# B&R Automation Studio project BuR
Automation Studio 4.5.2.102

## Logical view

### Package Logical/Libraries - Global libraries

### Library Logical/Libraries/DebuggingCom/DebComLib (IEC, version 1.00.1)
Depends on: astime, AsBrStr, TCPComLib

#### Types.typ - Exported data types
```iecst
TYPE
	e_DebugDataType : (E_STRING
		,E_DATA
	);

	e_DebugStepSend : (STEP_WAIT_FOR_ACTIVATE,
		STEP_WAIT_FOR_SEND_REQ,
		STEP_WAIT_FOR_ACK
	);

	s_SendDataType : STRUCT
		Data : ARRAY [0..ui_Max_Send_DataSize] OF BYTE;
		ui_Size : UINT;
	END_STRUCT;

	s_DebugDataType : STRUCT
		e_DataType : e_DebugDataType;
		ui_DataSize : UINT;
		(* *)
		tod_Time : TOD;
		dt_Date : DATE;
		str_Description : STRING[80];
		i_DataType : INT;
		aby_Data : ARRAY[0..ui_Data_Length_Pure_Data] OF BYTE;
    END_STRUCT;

	s_DebugDataBufferType : STRUCT
		Data : ARRAY[0..ui_Buffer_Size] OF s_DebugDataType;
        Size : INT := 0;
        Index : INT := 0;
	END_STRUCT;

    s_DebuggingComType : STRUCT
        b_init : BOOL := TRUE; (* Initialisierung *)
        b_Connected : BOOL;
        b_Error : BOOL;
        b_Enable_Com : BOOL := TRUE;
        Data : s_DebugDataBufferType;
        AddString : Add_Debug_String;
        AddData : Add_Debug_Data;
        TempStr : STRING[80];
        TempStr2 : STRING[80];
        Internal : s_DebugIternalType;
    END_STRUCT;

  s_DebugIternalType : STRUCT
    Cyclic : CyclicOperations;
  END_STRUCT;
END_TYPE
```

#### Constants.var - Exported constants
```iecst
VAR CONSTANT
	ui_Header_Length            : UINT := 6;          (* STX(1) + Laufnummer(1) + Trennbyte(1) + Telegrammtyp(2) + Trennbyte(1) *)
	ui_Footer_Length            : UINT := 1;          (* ETX(1) *)
	ui_Data_Length_String       : UINT := 90;         (* Zeit(4) + Trennbyte(1) + Datum(4) + Trennbyte(1) + Text(80) *)
	ui_Data_Length_Data         : UINT := 1449;       (* Zeit(4) + Trennbyte(1) + Datum(4) + Trennbyte(1) + Text(80) + Trennbyte(1) + Datentyp(2) + Trennbyte(1) + Daten(1355) *)
	ui_Data_Length_Pure_Data    : UINT := 1355;

	ui_SendDataLength_Debug     : UINT := ui_Header_Length + ui_Data_Length_String + ui_Footer_Length;
	ui_SendDataLength_Data      : UINT := ui_Header_Length + ui_Data_Length_Data + ui_Footer_Length;
	ui_RecDataLength_Quit       : UINT := ui_Header_Length + ui_Footer_Length; (* Quittierung erfolgt über Telegrammnummer *)

	ui_Max_Send_DataSize        : UINT := ui_SendDataLength_Data; (* Muss gröster Datenlänge entsprechen die gesendet werden soll *)

	ui_Buffer_Size              : UINT := 200; (* Größe des in der Steuerung gehaltenen Logs *)
END_VAR
```

#### DebComLib.fun - Exported functions and function blocks
```iecst
FUNCTION_BLOCK CyclicOperations (* *) (*$GROUP=User,$CAT=User,$GROUPICON=User.png,$CATICON=User.png*)
	VAR_INPUT
		Instance : REFERENCE TO s_DebuggingComType;
	END_VAR
	VAR
		FB_DebugCom : FBCom;
		DebugComConfig : s_FBComConfigType;
		FB_ConvertHeader    : ConvertHeader         ;
		FB_ConvertReceivedata : ConvertReceiveData  ;
		b_Enable           : BOOL                   ;
		b_Communicate       : BOOL  := FALSE        ;
		b_DataReceived       : BOOL                 ;
		b_AbortCommunication: BOOL                  ;
		b_Acknowledge      : BOOL                   ;
		b_Enable_Timeout   : BOOL                   ;
		b_Sending           : BOOL                  ;
		b_Wait_Ack          : BOOL                  ;
		b_Packet_Quit       : BOOL                  ;
		b_Data_Fail         : BOOL                  ;
		u16SendDataLength   : UINT                  ;
		u16ReceivedLength   : UDINT                 ;
		ui_pointer          : DINT                  ;
		ui_Packet_Length    : UINT                  ;
		ui_pointer_Data_in  : UINT                  ;
		i_Send_Versuche     : INT                   ;
		i_Rec_Versuche      : INT                   ;
		usi_Lfd_Nr_Send      : USINT                  ;
		usi_Lfd_Nr_Rec       : USINT                  ;
		rt_Count_Send       : R_TRIG                ;
        ton_SendCycle       : TON                   ;
        i_Temp              : INT                   ;

		e_StepSend         : e_DebugStepSend        ;
		e_OldStepSend      : e_DebugStepSend        ;

		aby_SendBuffer : ARRAY [0..ui_Max_Send_DataSize] OF BYTE;
		aby_ReceiveBuffer : ARRAY [0..ui_RecDataLength_Quit] OF BYTE;
		aby_TempBuffer : ARRAY [0..ui_RecDataLength_Quit] OF BYTE;
		aby_Temp : ARRAY[0..ui_Max_Send_DataSize] OF BYTE;
	END_VAR
END_FUNCTION_BLOCK

FUNCTION_BLOCK Add_Debug_String (*//======= Add_Debug_String ===========================================================
// Funktion         : Diese Funktion fügt einen neuen Text und die aktuelle Zeit zum Puffer hinzu
//
// Eingansparameter :
//               str_Text            : zu schreibender Text (STRING[80])
//
// Rückgabewert :
//
// Unterprogramme   : keine
//
// Benötigte Units  :
//
// Aenderungen      :
//
// Aenderungsdatum  :
//
//----------------------------------------------------------------------------------------*) (*$GROUP=User,$CAT=User,$GROUPICON=User.png,$CATICON=User.png*)
	VAR_INPUT
		Instance : REFERENCE TO s_DebuggingComType;
		str_Text : STRING[80];
	END_VAR
	VAR
        realtime : DTStructureGetTime;
		ActTime : DTStructure;
	END_VAR
END_FUNCTION_BLOCK

FUNCTION_BLOCK Add_Debug_Data (*//======= Add_Debug_Data ===========================================================
// Funktion         : Diese Funktion fügt einen neuen Text, neue Daten und die aktuelle Zeit zum Puffer hinzu
//
// Eingansparameter :
//               str_Text            : zu schreibender Text (STRING[80])
//               i_DataType          : Datentyp in aby_Data (INT)
//               aby_Data            : Daten (ARRAY[0..1372] OF BYTE)
//               ui_DataSize         : Länge der übergebenen Daten (UINT)
//
// Rückgabewert :
//
// Unterprogramme   : keine
//
// Benötigte Units  :
//
// Aenderungen      :
//
// Aenderungsdatum  :
//
//----------------------------------------------------------------------------------------*) (*$GROUP=User,$CAT=User,$GROUPICON=User.png,$CATICON=User.png*)
	VAR_INPUT
		Instance : REFERENCE TO s_DebuggingComType;
		str_Text : STRING[80];
		i_DataType : INT;
		aby_Data : ARRAY[0..ui_Data_Length_Pure_Data] OF BYTE;
		ui_DataSize : UINT;
	END_VAR
	VAR
        realtime : DTStructureGetTime;
		ActTime : DTStructure;
	END_VAR
END_FUNCTION_BLOCK

FUNCTION MakeData : USINT
	(*//======= MakeData ===========================================================
	// Funktion         : Diese Funktion konvertiert den Debugtext in ein Bytearray
	//
	// Eingansparameter :
	//
	// Durchgangsparameter :
	//               Data            : Datengrundlage (s_DebugDataType)
	//           aby_Result          : Ergebnis (ARRAY[0..ui_Max_Send_DataSize-1] OF BYTE)
	//
	// Rückgabewert :
	//
	// Unterprogramme   : keine
	//
	// Benötigte Units  :
	//
	// Aenderungen      :
	//
	// Aenderungsdatum  :
	//
	//----------------------------------------------------------------------------------------*)

	VAR_IN_OUT
		Data : s_DebugDataType; (* Datengrundlage *)
		aby_Result : ARRAY[0..ui_Max_Send_DataSize] OF BYTE; (* Ergebnis *)
	END_VAR

	VAR
		i_Temp : INT;
		by_Temp : BYTE;
		tod_Temp : TIME_OF_DAY;
		udi_Temp : UDINT;
	END_VAR

		END_FUNCTION

FUNCTION GetNextTelegramNo : USINT
	VAR_IN_OUT
		usi_ActNo : USINT;
	END_VAR
		END_FUNCTION

FUNCTION MakeSendData : USINT
	(*//======= MakeSendData ===========================================================
	// Funktion         : Diese Funktion setzt den Header und Footer an die Nutdaten
	//
	// Eingansparameter :
	//               ui_DataLength      : genutzte Übergabedatenlänge (UINT)
	//               usi_lfd_Nr         : Telegrammlaufnummer (USINT)
	//
	// Durchgangsparameter :
	//               aby_SourceData     : Datenarray (ARRAY[0..ui_Max_Send_DataSize] OF BYTE)
	//               aby_Result         : Datenarray (ARRAY[0..ui_Max_Send_DataSize - 1] OF BYTE)
	//
	// Rückgabewert :
	//
	// Unterprogramme   : keine
	//
	// Benötigte Units  :
	//
	// Aenderungen      :
	//
	// Aenderungsdatum  :
	//
	//----------------------------------------------------------------------------------------*)
	VAR_INPUT
		ui_DataLength : UINT;
		usi_lfd_Nr : USINT;
		i_TelegrammType : INT;
	END_VAR

	VAR_IN_OUT
		aby_SourceData : ARRAY[0..ui_Max_Send_DataSize] OF BYTE;
		aby_Result : ARRAY[0..ui_Max_Send_DataSize] OF BYTE;
	END_VAR

	VAR
		by_Temp     : BYTE;
		i_Temp : INT;
	END_VAR
			END_FUNCTION

FUNCTION_BLOCK ConvertHeader
	(*//======= ConvertHeader ===========================================================
	// Funktion         : Dieser Funktionsbaustein prüft die empfangenen Headerdaten
	//                 Gibt notwendige Headerdaten aus
	//
	// Eingansparameter :
	//
	// Ein- Ausgansparameter :
	//                   aby_SourceData     : Datenarray (ARRAY[0..ui_RecDataLength_Quit] OF BYTE)
	//
	// Ausgangsparameter:
	//             usi_lfd_Nr_Rec       : Telegrammlaufnummer (USINT)
	//             i_Telegramm_Nr       : Nummer des empfangenen Telegramms (INT)
	//             ui_TotalDataLength   : erwartete Gesammtdatenmenge (UINT)
	//             b_Data_Ok            : Daten Ok (BOOL)
	//
	// Unterprogramme   : keine
	//
	// Benötigte Units  :
	//
	// Aenderungen      :
	//
	// Aenderungsdatum  :
	//
	//----------------------------------------------------------------------------------------*)
	VAR_IN_OUT
		aby_SourceData : ARRAY[0..ui_RecDataLength_Quit] OF BYTE;
	END_VAR

	VAR_OUTPUT
		usi_lfd_Nr_Rec : USINT;
		i_Telegramm_Nr : INT;
		ui_TotalDataLength : UINT;
		b_Data_Ok : BOOL;
	END_VAR

	VAR
		i_Temp : INT;
	END_VAR

		END_FUNCTION_BLOCK

FUNCTION_BLOCK ConvertReceiveData
	(*//======= ConvertReceiveData ===========================================================
	// Funktion         : Dieser Funktionsbaustein prüft die empfangenen Daten
	//                 Entfernt Header und Footer
	//                 Gibt notwendige Daten aus
	//
	//
	// Eingansparameter :
	//               ui_DataLength      : übergebene Nutzdatenlänge (UINT)
	//               i_Telegramm_Nr       : Nummer des empfangenen Telegramms (INT)
	//
	// Ein- Ausgansparameter :
	//
	// Ausgangsparameter:
	//               b_Data_Ok          : Daten sind ok (BOOL);
	//
	//
	// Unterprogramme   : keine
	//
	// Benötigte Units  :
	//
	// Aenderungen      :
	//
	// Aenderungsdatum  :
	//
	//----------------------------------------------------------------------------------------*)
	VAR_INPUT
		ui_DataLength : UINT;
		i_Telegramm_Nr : INT;
	END_VAR

	VAR_OUTPUT
		b_Data_Ok : BOOL;
	END_VAR

		END_FUNCTION_BLOCK
```

#### CyclicOperations.st
```iecst
(* TODO: Hier einen Kommentar eingeben *)
FUNCTION_BLOCK CyclicOperations

	IF Instance.b_init THEN
		DebugComConfig.Connection.b_IsClient := FALSE;
		DebugComConfig.Connection.ui_LocalPort := 5000;
		usi_Lfd_Nr_Send := 0;
		i_Send_Versuche := 0;
		i_Rec_Versuche := 0;

		Instance.b_init := FALSE;
	END_IF;

	CASE e_StepSend OF

		STEP_WAIT_FOR_ACTIVATE:

			IF b_AbortCommunication THEN
				b_AbortCommunication  := FALSE;
			END_IF;

			b_Acknowledge := FALSE;
			b_Communicate := FALSE;
			usi_Lfd_Nr_Send := 0;

			IF b_Enable AND Instance.b_Connected THEN
				e_StepSend := STEP_WAIT_FOR_SEND_REQ;
			END_IF;

		STEP_WAIT_FOR_SEND_REQ:

			// Flankenerzeugung
			b_Communicate      := FALSE;
			b_Acknowledge      := FALSE;

			IF NOT b_Enable THEN
				// Kommunikation deaktivieren

				e_StepSend := STEP_WAIT_FOR_ACTIVATE;
			ELSIF NOT Instance.b_Connected THEN
				// Verbindung wurde geschlossen

				e_StepSend := STEP_WAIT_FOR_ACTIVATE;
			ELSIF b_AbortCommunication THEN
				b_AbortCommunication  := FALSE;
				b_Acknowledge := FALSE;

			ELSE
                IF NOT b_Sending AND NOT b_Communicate AND NOT b_Wait_Ack AND Instance.Data.Size > 0 THEN
                    i_Temp := (Instance.Data.Index + (-(Instance.Data.Size) + ui_Buffer_Size)) MOD ui_Buffer_Size;
                    MakeData(
					Data := Instance.Data.Data[i_Temp]
					,aby_Result := aby_Temp
					);

					IF Instance.Data.Data[i_Temp].e_DataType = E_STRING THEN
						MakeSendData(
							ui_DataLength := ui_Data_Length_String
							,usi_lfd_Nr := GetNextTelegramNo(usi_Lfd_Nr_Send)
							,i_TelegrammType := 16#3032
							,aby_SourceData := aby_Temp
							,aby_Result := aby_SendBuffer
							);
						u16SendDataLength := ui_SendDataLength_Debug;
					ELSE
						MakeSendData(
							ui_DataLength := ui_Data_Length_Data
							,usi_lfd_Nr := GetNextTelegramNo(usi_Lfd_Nr_Send)
							,i_TelegrammType := 16#3033
							,aby_SourceData := aby_Temp
							,aby_Result := aby_SendBuffer
							);
						u16SendDataLength := ui_SendDataLength_Data;
					END_IF;

					b_Communicate := TRUE;
					b_Wait_Ack := TRUE;

					Instance.Data.Size := Instance.Data.Size - 1;

					e_StepSend := STEP_WAIT_FOR_ACK;
				ELSIF b_Wait_Ack THEN
					b_Communicate := TRUE;

					e_StepSend := STEP_WAIT_FOR_ACK;
				END_IF;
			END_IF;

		STEP_WAIT_FOR_ACK:

			// Flankenerzeugung
			b_Communicate := FALSE;

			IF ton_SendCycle.Q THEN
				b_Communicate := TRUE;
			END_IF;

			IF NOT b_Enable THEN
				// Kommunikation deaktivieren

				e_StepSend := STEP_WAIT_FOR_ACTIVATE;
			ELSIF b_AbortCommunication THEN
				// aktuellen Übertragungsvorgang abbrechen

				e_StepSend := STEP_WAIT_FOR_SEND_REQ;
			ELSIF NOT Instance.b_Connected THEN
				// Verbindung wurde geschlossen

				e_StepSend := STEP_WAIT_FOR_ACTIVATE;
			ELSE
				// Quittung empfangen -> auswerten
				IF b_Packet_Quit THEN
					b_Acknowledge := TRUE;
					b_Wait_Ack := FALSE;
					b_Packet_Quit := FALSE;

					e_StepSend := STEP_WAIT_FOR_SEND_REQ;
				END_IF;

			END_IF;

		ELSE
			;
	END_CASE;

	// Timer für zyklisches "Neu-Senden", falls keine Quittung innerhalb der konfigurierten Wartezeit kommt
	b_Enable_Timeout := (e_StepSend = STEP_WAIT_FOR_ACK) AND
	e_StepSend = e_OldStepSend;

	ton_SendCycle (IN := b_Enable_Timeout AND NOT b_Communicate AND NOT ton_SendCycle.Q, PT := t#2000ms);
	e_OldStepSend := e_StepSend;

	// Zähler Sendeversuche
	rt_Count_Send (CLK := b_Sending AND e_StepSend = STEP_WAIT_FOR_ACK); // Flanke zählen Sendeversuche

	// Zähler Rücksetzen
	IF b_Acknowledge OR NOT b_Enable THEN
		i_Send_Versuche := 0;
	END_IF;

	// Zähler Empfangsversuche
	IF b_Data_Fail THEN
		i_Rec_Versuche := i_Rec_Versuche + 1;
	END_IF;

	// Zähler Rücksetzen
	IF NOT b_Enable THEN
		i_Rec_Versuche := 0;
	END_IF;

	IF Instance.b_Enable_Com AND NOT Instance.b_init AND i_Send_Versuche <= 3 AND i_Rec_Versuche <= 3 AND NOT FB_DebugCom.error THEN
		b_Enable := TRUE ;
	ELSE
		b_Enable := FALSE ;
		ui_pointer_Data_in := 0;
	END_IF ;

	//call communication function block
	FB_DebugCom(
		enable := b_Enable
		,send := b_Communicate
		,sendDataLength := u16SendDataLength
		,receiveDataLength := SIZEOF(aby_ReceiveBuffer)
		,configurations := DebugComConfig
		,sendBuffer := ADR(aby_SendBuffer)
		,receiveBuffer := ADR(aby_ReceiveBuffer)
	);
	u16ReceivedLength := FB_DebugCom.receivedDataLength;
	Instance.b_Connected := FB_DebugCom.connected;
	b_DataReceived := FB_DebugCom.dataReceived;
	b_Sending := FB_DebugCom.sending;

	b_Data_Fail := FALSE;

	IF Instance.b_Connected THEN
		// Wenn richtige Datenlänge empfangen und in Speicher eintragen
		IF b_DataReceived THEN
			FOR ui_pointer := 0 TO UDINT_TO_DINT(u16ReceivedLength) - 1 DO

				aby_TempBuffer[ui_pointer_Data_in] := aby_ReceiveBuffer[ui_pointer] ;
				ui_pointer_Data_in := ui_pointer_Data_in + 1;

				IF ui_pointer_Data_in = ui_Header_Length THEN
					FB_ConvertHeader(
						aby_SourceData := aby_TempBuffer
						//,usi_Lfd_Nr_Rec =>
						// ,i_Telegramm_Nr =>
						//,ui_TotalDataLength =>
						// ,b_Data_Ok
						);
					usi_Lfd_Nr_Rec := FB_ConvertHeader.usi_lfd_Nr_Rec;
					ui_Packet_Length := FB_ConvertHeader.ui_TotalDataLength;
				END_IF;

				// Unbekannte Telegrammnummer
				IF ui_pointer_Data_in = ui_Header_Length AND NOT FB_ConvertHeader.b_Data_Ok THEN
					b_Data_Fail := TRUE;
					ui_pointer_Data_in := 0;
				END_IF;

				IF ui_pointer_Data_in = ui_Packet_Length AND ui_pointer_Data_in > ui_Header_Length THEN
					IF aby_TempBuffer[ui_pointer_Data_in - 1] = 16#03 THEN
						// Ende Datenstream
						FB_ConvertReceivedata(
							ui_DataLength := ui_Packet_Length
						,i_Telegramm_Nr := FB_ConvertHeader.i_Telegramm_Nr
						// ,b_Data_Ok =>
						);
						CASE FB_ConvertReceivedata.i_Telegramm_Nr OF

							11: b_Packet_Quit := FB_ConvertHeader.b_Data_Ok AND FB_ConvertReceivedata.b_Data_Ok;

							12: b_Packet_Quit := FB_ConvertHeader.b_Data_Ok AND FB_ConvertReceivedata.b_Data_Ok;

							13: b_Packet_Quit := FB_ConvertHeader.b_Data_Ok AND FB_ConvertReceivedata.b_Data_Ok;

						END_CASE;
						ui_pointer_Data_in := 0 ;
						i_Rec_Versuche := 0;
					ELSE
						ui_pointer_Data_in := 0 ;
						b_Data_Fail := TRUE;
					END_IF;
				END_IF;
			END_FOR ;
		END_IF ;
	ELSE
		ui_pointer_Data_in := 0 ;
	END_IF;

END_FUNCTION_BLOCK
```

#### AddDebugString.st
```iecst
FUNCTION_BLOCK Add_Debug_String
    realtime(enable := TRUE, pDTStructure := ADR(ActTime));
    Instance.Data.Data[Instance.Data.Index].e_DataType := E_STRING;
    Instance.Data.Data[Instance.Data.Index].ui_DataSize := 0;
    Instance.Data.Data[Instance.Data.Index].tod_Time := DT_TO_TOD(DTStructure_TO_DT(ADR(ActTime))) + UINT_TO_TIME(ActTime.millisec);
    Instance.Data.Data[Instance.Data.Index].dt_Date := DT_TO_DATE(DTStructure_TO_DT(ADR(ActTime)));
    Instance.Data.Data[Instance.Data.Index].str_Description := str_Text;
    Instance.Data.Data[Instance.Data.Index].i_DataType := -1;
    Instance.Data.Index := (Instance.Data.Index + 1) MOD ui_Buffer_Size;
    Instance.Data.Size :=  MIN(Instance.Data.Size + 1, UINT_TO_INT(ui_Buffer_Size));
END_FUNCTION_BLOCK
```

#### AddDebugData.st
```iecst
FUNCTION_BLOCK Add_Debug_Data
	realtime(enable := TRUE, pDTStructure := ADR(ActTime));
    Instance.Data.Data[Instance.Data.Index].e_DataType := E_DATA;
	Instance.Data.Data[Instance.Data.Index].ui_DataSize := MIN(ui_DataSize, ui_Data_Length_Pure_Data) ;
	Instance.Data.Data[Instance.Data.Index].tod_Time := DT_TO_TOD(DTStructure_TO_DT(ADR(ActTime))) + UINT_TO_TIME(ActTime.millisec);
	Instance.Data.Data[Instance.Data.Index].dt_Date := DT_TO_DATE(DTStructure_TO_DT(ADR(ActTime)));
	Instance.Data.Data[Instance.Data.Index].str_Description := str_Text;
	Instance.Data.Data[Instance.Data.Index].i_DataType := i_DataType;
	Instance.Data.Data[Instance.Data.Index].aby_Data := aby_Data;
    Instance.Data.Index := (Instance.Data.Index + 1) MOD ui_Buffer_Size;
    Instance.Data.Size :=  MIN(Instance.Data.Size + 1, UINT_TO_INT(ui_Buffer_Size));
END_FUNCTION_BLOCK
```

#### InternalFunctions.st
```iecst
FUNCTION MakeData
	// Reset memory data
	brsmemset(ADR(aby_Result[0]), 0, SIZEOF(aby_Result));
	// Zeit
	tod_Temp := swapTOD(H_TO_NTOD(Data.tod_Time));
	brsmemcpy(ADR(aby_Result[0]), ADR(tod_Temp), SIZEOF(tod_Temp));
	// Trennbyte
	by_Temp := 16#2e;
	brsmemcpy(ADR(aby_Result[4]), ADR(by_Temp), SIZEOF(by_Temp));
	// Datum (convert to days since 01.01.1992)
	udi_Temp := swapUDINT(H_TO_NUDINT((DATE_TO_UDINT(Data.dt_Date) - DATE_TO_UDINT(D#1992-01-01)) / 86400));
	brsmemcpy(ADR(aby_Result[5]), ADR(udi_Temp), SIZEOF(udi_Temp));
	// Trennbyte
	by_Temp := 16#2e;
	brsmemcpy(ADR(aby_Result[9]), ADR(by_Temp), SIZEOF(by_Temp));
	// Text
	brsmemcpy(ADR(aby_Result[10]), ADR(Data.str_Description), brsstrlen(ADR(Data.str_Description)));

	IF Data.e_DataType = E_DATA THEN
		// Trennbyte
		by_Temp := 16#2e;
		brsmemcpy(ADR(aby_Result[90]), ADR(by_Temp), SIZEOF(by_Temp));
		// Datentyp
		i_Temp := swapINT(H_TO_NINT(Data.i_DataType));
		brsmemcpy(ADR(aby_Result[91]), ADR(i_Temp), SIZEOF(i_Temp));
		// Trennbyte
		by_Temp := 16#2e;
		brsmemcpy(ADR(aby_Result[93]), ADR(by_Temp), SIZEOF(by_Temp));
		// Daten
		brsmemcpy(ADR(aby_Result[94]), ADR(Data.aby_Data), Data.ui_DataSize);
    END_IF;
    MakeData := 0;

END_FUNCTION

FUNCTION GetNextTelegramNo

	usi_ActNo := (usi_ActNo MOD 255) + 1;
	GetNextTelegramNo := usi_ActNo;
END_FUNCTION

FUNCTION MakeSendData

	// Reset memory data
	brsmemset(ADR(aby_Result[0]), 0, SIZEOF(aby_Result));
	// Startzeichen
	by_Temp := 16#02;
	brsmemcpy(ADR(aby_Result[0]), ADR(by_Temp), SIZEOF(by_Temp));
	// Telegrammlaufnummer
	brsmemcpy(ADR(aby_Result[1]), ADR(usi_lfd_Nr), SIZEOF(usi_lfd_Nr));
	// Trennbyte
	by_Temp := 16#2E;
	brsmemcpy(ADR(aby_Result[2]), ADR(by_Temp), SIZEOF(by_Temp));
	// Telegrammtyp
	i_Temp := H_TO_NINT(i_TelegrammType);
	brsmemcpy(ADR(aby_Result[3]), ADR(i_Temp), SIZEOF(i_TelegrammType));
	// Trennbyte
	by_Temp := 16#2E;
	brsmemcpy(ADR(aby_Result[5]), ADR(by_Temp), SIZEOF(by_Temp));
	// Daten einfügen
	brsmemcpy(ADR(aby_Result[6]), ADR(aby_SourceData), ui_DataLength);

	// Endzeichen
    aby_Result[MIN(ui_DataLength + 6, ui_Max_Send_DataSize)] := 16#03;

    MakeSendData := 0;
END_FUNCTION

FUNCTION_BLOCK ConvertHeader

	//Telegrammlaufnummer
	brsmemcpy(ADR(usi_lfd_Nr_Rec), ADR(aby_SourceData[1]), SIZEOF(usi_lfd_Nr_Rec));

	// Telegrammnummer
	brsmemcpy(ADR(i_Temp), ADR(aby_SourceData[3]), SIZEOF(i_Temp));
	i_Temp := N_TO_HINT(i_Temp);

	i_Telegramm_Nr := 0;
	ui_TotalDataLength := 0;

	CASE i_Temp OF

		16#3130:

		ui_TotalDataLength := ui_RecDataLength_Quit;
		i_Telegramm_Nr := 10;
		b_Data_Ok := TRUE;

		16#3131:

		ui_TotalDataLength := ui_RecDataLength_Quit;
		i_Telegramm_Nr := 11;
		b_Data_Ok := TRUE;

		16#3132:

		ui_TotalDataLength := ui_RecDataLength_Quit;
		i_Telegramm_Nr := 12;
		b_Data_Ok := TRUE;

		16#3133:

		ui_TotalDataLength := ui_RecDataLength_Quit;
		i_Telegramm_Nr := 13;
		b_Data_Ok:= TRUE;

		ELSE

			b_Data_Ok := FALSE;

	END_CASE;
END_FUNCTION_BLOCK

FUNCTION_BLOCK ConvertReceiveData

	b_Data_Ok := TRUE;
	CASE i_Telegramm_Nr OF

		10:

			b_Data_Ok := b_Data_Ok AND (ui_DataLength = ui_RecDataLength_Quit);

		11:

			b_Data_Ok := b_Data_Ok AND (ui_DataLength = ui_RecDataLength_Quit);

		12:

			b_Data_Ok := b_Data_Ok AND (ui_DataLength = ui_RecDataLength_Quit);

		13:

			b_Data_Ok := b_Data_Ok AND (ui_DataLength = ui_RecDataLength_Quit);

		ELSE
			b_Data_Ok := FALSE;
	END_CASE;

END_FUNCTION_BLOCK
```

### Program Logical/Libraries/DebuggingCom/DebugComCycle (IEC)

#### Types.typ
```iecst
TYPE

	e_DebugStepType : (E_DBST_WAIT_FOR_ACTIVATE
	);

END_TYPE
```

#### Main.st
```iecst
PROGRAM _INIT
	DebuggingCom.b_init := TRUE;
	DebuggingCom.Internal.Cyclic.Instance := ADR(DebuggingCom);
	DebuggingCom.AddString.Instance := ADR(DebuggingCom);
	DebuggingCom.AddData.Instance := ADR(DebuggingCom);
END_PROGRAM

PROGRAM _CYCLIC

	DebuggingCom.Internal.Cyclic();

END_PROGRAM

PROGRAM _EXIT

END_PROGRAM
```
